(* Low pass Infinite Impulse Response (IIR) filter*)
FUNCTION_BLOCK InfiniteImpulseResponse IMPLEMENTS IOut
VAR_INPUT
    new : LREAL;
    decay : LREAL;
END_VAR
VAR
    _previous : LREAL;
    _out : LREAL;
END_VAR

_out := _previous * decay + new * (1 - decay);
_previous := _out;

PROPERTY Out : LREAL
GET
Out := _out;
END_GET
END_PROPERTY

END_FUNCTION_BLOCK

(* stored: Version 1.1.0.1
   POU InfiniteImpulseResponse: Id {f8c814fe-9c50-4fa3-be31-ddba18f7ea5c}, SpecialFunc None
   Property Out: Id {0947fad0-a47b-4436-9f1f-02025124f8a9}
   Get Get: Id {a19f5262-6b95-469f-bc31-d14a4bf3fb97} *)
